% RSLogix 500 project Proyecto2_Cajas.RSS, saved by version 8.30.00.16 %
PROJECT "UNTITLED"    % processor: Bul.1763 MicroLogix 1100 Series B %

PROGRAM FILES
  LAD 2   3 rungs
  LAD 3 "DIGITAL IO"  8 rungs
  LAD 4 "CONTROL"  6 rungs

DATA FILES
  O0 OUTPUT  4 elements
  I1 INPUT  6 elements
  S2 STATUS  66 elements
  B3 BINARY  3 elements
  T4 TIMER  2 elements
  C5 COUNTER  1 elements
  R6 CONTROL  1 elements
  N7 INTEGER  1 elements
  F8 FLOAT  1 elements

LADDER 2
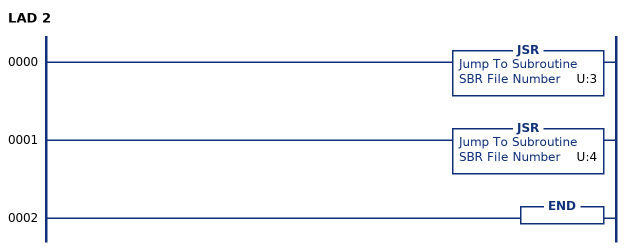
% Rung: 0 %
SOR JSR U:3 EOR
% Rung: 1 %
SOR JSR U:4 EOR
% Rung: 2 %
SOR END EOR

LADDER 3 "DIGITAL IO"
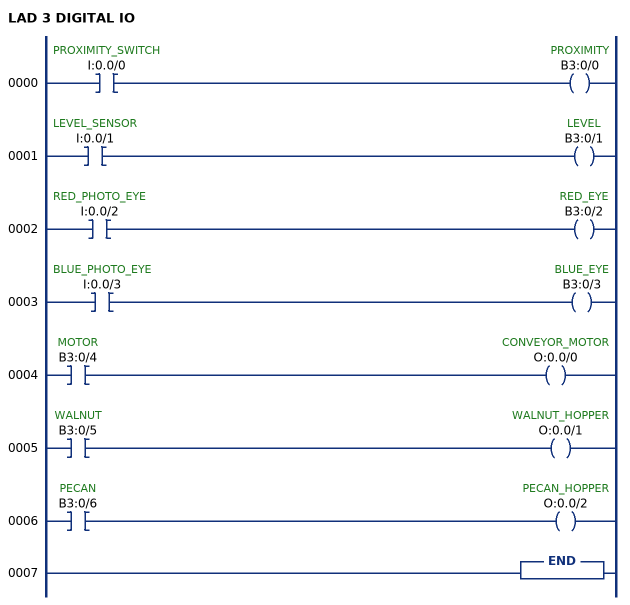
% Rung: 0 %
SOR XIC I:0.0/0 OTE B3:0/0 EOR
%   I:0.0/0  PROXIMITY_SWITCH %
%   B3:0/0  PROXIMITY %
% Rung: 1 %
SOR XIC I:0.0/1 OTE B3:0/1 EOR
%   I:0.0/1  LEVEL_SENSOR %
%   B3:0/1  LEVEL %
% Rung: 2 %
SOR XIC I:0.0/2 OTE B3:0/2 EOR
%   I:0.0/2  RED_PHOTO_EYE %
%   B3:0/2  RED_EYE %
% Rung: 3 %
SOR XIC I:0.0/3 OTE B3:0/3 EOR
%   I:0.0/3  BLUE_PHOTO_EYE %
%   B3:0/3  BLUE_EYE %
% Rung: 4 %
SOR XIC B3:0/4 OTE O:0.0/0 EOR
%   B3:0/4  MOTOR %
%   O:0.0/0  CONVEYOR_MOTOR %
% Rung: 5 %
SOR XIC B3:0/5 OTE O:0.0/1 EOR
%   B3:0/5  WALNUT %
%   O:0.0/1  WALNUT_HOPPER %
% Rung: 6 %
SOR XIC B3:0/6 OTE O:0.0/2 EOR
%   B3:0/6  PECAN %
%   O:0.0/2  PECAN_HOPPER %
% Rung: 7 %
SOR END EOR

LADDER 4 "CONTROL"
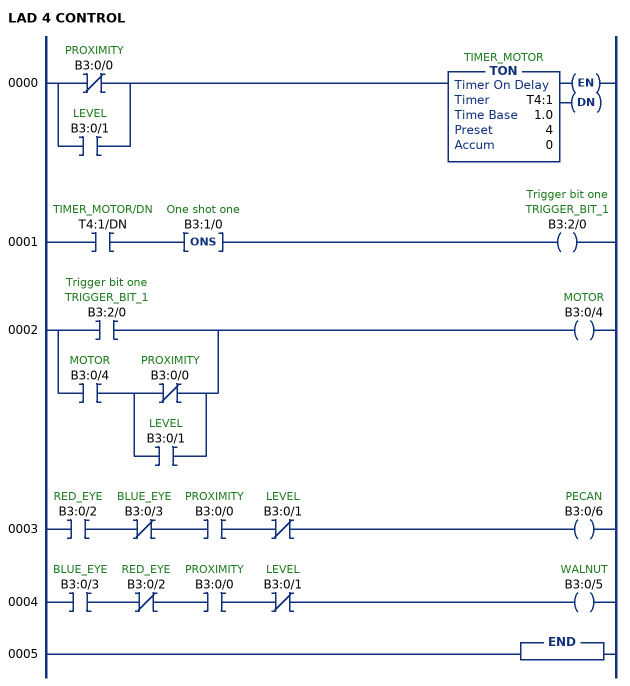
% Rung: 0 %
SOR BST XIO B3:0/0 NXB XIC B3:0/1 BND TON T4:1 1.0 4 0 EOR
%   B3:0/0  PROXIMITY %
%   B3:0/1  LEVEL %
%   T4:1  TIMER_MOTOR %
% Rung: 1 %
SOR XIC T4:1/DN ONS B3:1/0 OTE B3:2/0 EOR
%   T4:1  TIMER_MOTOR %
%   B3:1/0  "One shot one" %
%   B3:2/0  TRIGGER_BIT_1  "Trigger bit one" %
% Rung: 2 %
SOR BST XIC B3:2/0 NXB XIC B3:0/4 BST XIO B3:0/0 NXB XIC B3:0/1 BND BND OTE B3:0/4 EOR
%   B3:2/0  TRIGGER_BIT_1  "Trigger bit one" %
%   B3:0/4  MOTOR %
%   B3:0/0  PROXIMITY %
%   B3:0/1  LEVEL %
% Rung: 3 %
SOR XIC B3:0/2 XIO B3:0/3 XIC B3:0/0 XIO B3:0/1 OTE B3:0/6 EOR
%   B3:0/2  RED_EYE %
%   B3:0/3  BLUE_EYE %
%   B3:0/0  PROXIMITY %
%   B3:0/1  LEVEL %
%   B3:0/6  PECAN %
% Rung: 4 %
SOR XIC B3:0/3 XIO B3:0/2 XIC B3:0/0 XIO B3:0/1 OTE B3:0/5 EOR
%   B3:0/3  BLUE_EYE %
%   B3:0/2  RED_EYE %
%   B3:0/0  PROXIMITY %
%   B3:0/1  LEVEL %
%   B3:0/5  WALNUT %
% Rung: 5 %
SOR END EOR

DATA TABLE (non-zero values as saved)
DATA T4
% .PRE .ACC %
% T4:1 % 4 0
